(* Logix 5000 project; controller cal1632 1756-L62 rev 16.20; software revision 16.05; part 55 of 57 *)
(* tags used below, declared in another part *)
   FAULT : BOOL;
   p01_recipe_active : recipe;
   p01r02_plc_scan_time_in_sec : REAL;
   p01r09_pb_global_reset : BOOL;
   p29_ao_wdr_turret_selected_speed : REAL;
   p29_di_turret_pos : BOOL;
   p29_di_wdr_index_fwd : BOOL;
   p29_di_wdr_turret : acs800_di_normal;
   p29_di_wt_motor : BOOL;
   p29_do_wdr_turret : acs800_do_normal;
   p29_param_fast_turret_speed : REAL;
   p29_param_slow_turret_speed : REAL;
   p29r15_wdra_active : BOOL;
   p29r16_wdrb_active : BOOL;
   p29r20 : routine;
   p29r20_acc_dec_ramp : SYS_ACC_DEC_RAMP;
   p29r20_accel_rate : REAL;
   p29r20_decel_rate : REAL;
   p29r20_fast_accel : REAL;
   p29r20_fast_decel : REAL;
   p29r20_index_complete : BOOL;
   p29r20_index_move_timer : TIMER;
   p29r20_permissive : BOOL;
   p29r20_request_fwd : BOOL;
   p29r20_request_rev : BOOL;
   p29r20_selected_speed : REAL;
   p29r20_timer_fault : TIMER[10];
   p29r20_timer_warning : TIMER[4];
   p29r20_zero_speed : BOOL;
   p30_di_pin_1 : BOOL;
   p30_di_pin_2 : BOOL;
   p30_di_pin_3 : BOOL;
   p30_di_pin_4 : BOOL;
   p30_di_pin_5 : BOOL;
   p30_di_pin_6 : BOOL;
   p30_di_pin_7 : BOOL;
   p30_di_pin_8 : BOOL;
   p30_di_retraction_down_ls : BOOL;
   p30_di_retraction_up_ls : BOOL;
   p30_di_rotation_fault : BOOL;
   p30_di_ss_close : BOOL;
   p30_di_ss_open : BOOL;
   p30_dint_to_hmi : DINT[16];
   p30r01 : routine;
   p30r02 : routine;
   p30r02_fault_exists : BOOL;
   p30r02_timer_fault : TIMER[4];
   p30r02_timer_warning : TIMER[4];
   p30r02_unack_fault : BOOL;
   p30r02_unack_warning : BOOL;
   p30r02_warning_exists : BOOL;
   p30r03 : routine;
   p30r03_timer_fault : TIMER[4];
   p30r03_timer_warning : TIMER[4];
   p30r04 : routine;
   p30r05 : routine;
   p30r06 : routine;
   p30r07 : routine;
   p30r08 : routine;
   p30r09 : routine;
   p30r10 : routine;
   RETACTION_DELAY_TIMER : TIMER;
   RETRACTION_DELAY_TIMER_2 : TIMER;
(* P29_Winder, continued *)

ROUTINE R20_Winder_Turret_VFD   (* ladder *)
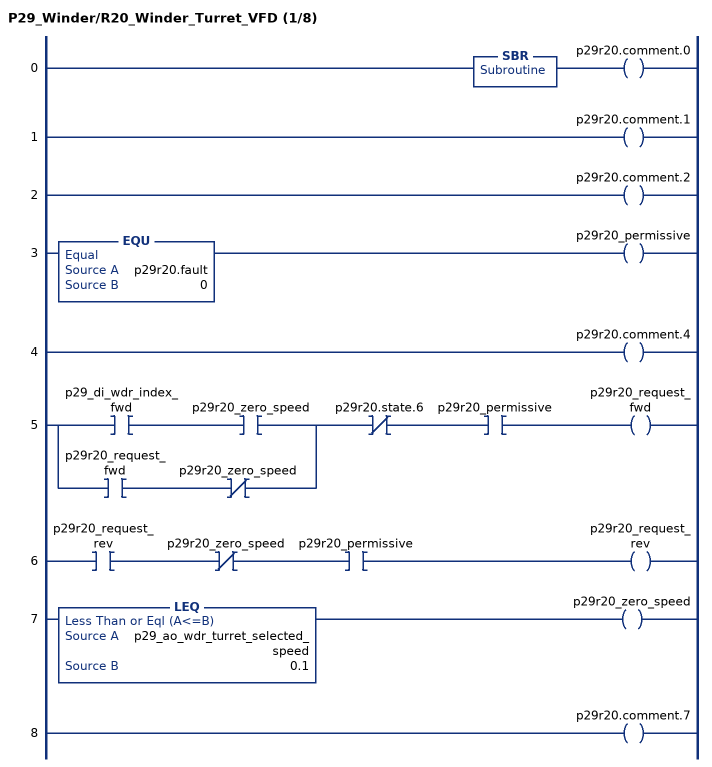
   0: SBR()OTE(p29r20.comment.0);
   1: OTE(p29r20.comment.1);
   2: OTE(p29r20.comment.2);
   3: EQU(p29r20.fault,0)OTE(p29r20_permissive);
   4: OTE(p29r20.comment.4);
   5: [XIC(p29_di_wdr_index_fwd) XIC(p29r20_zero_speed) ,XIC(p29r20_request_fwd) XIO(p29r20_zero_speed) ]XIO(p29r20.state.6)XIC(p29r20_permissive)OTE(p29r20_request_fwd);
   6: XIC(p29r20_request_rev)XIO(p29r20_zero_speed)XIC(p29r20_permissive)OTE(p29r20_request_rev);
   7: LEQ(p29_ao_wdr_turret_selected_speed,0.1)OTE(p29r20_zero_speed);
   8: OTE(p29r20.comment.7);
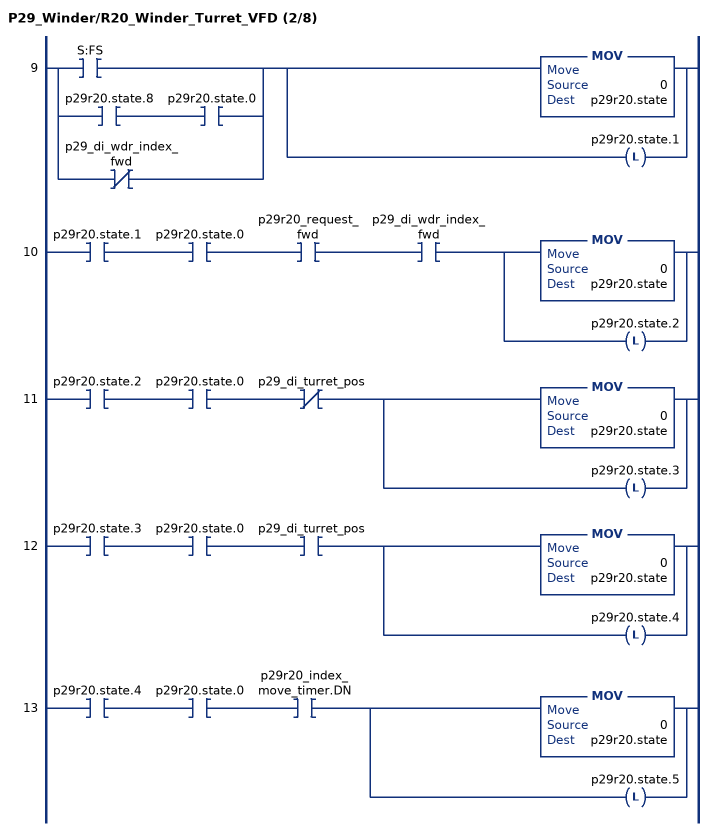
   9: [XIC(S:FS) ,XIC(p29r20.state.8) XIC(p29r20.state.0) ,XIO(p29_di_wdr_index_fwd) ][MOV(0,p29r20.state) ,OTL(p29r20.state.1) ];
   10: XIC(p29r20.state.1)XIC(p29r20.state.0)XIC(p29r20_request_fwd)XIC(p29_di_wdr_index_fwd)[MOV(0,p29r20.state) ,OTL(p29r20.state.2) ];
   11: XIC(p29r20.state.2)XIC(p29r20.state.0)XIO(p29_di_turret_pos)[MOV(0,p29r20.state) ,OTL(p29r20.state.3) ];
   12: XIC(p29r20.state.3)XIC(p29r20.state.0)XIC(p29_di_turret_pos)[MOV(0,p29r20.state) ,OTL(p29r20.state.4) ];
   13: XIC(p29r20.state.4)XIC(p29r20.state.0)XIC(p29r20_index_move_timer.DN)[MOV(0,p29r20.state) ,OTL(p29r20.state.5) ];
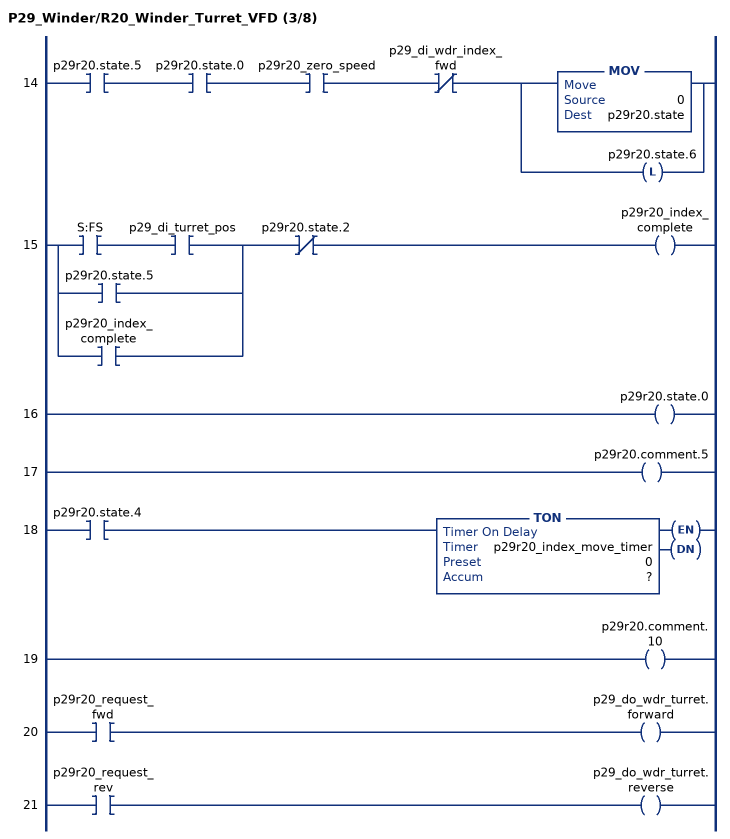
   14: XIC(p29r20.state.5)XIC(p29r20.state.0)XIC(p29r20_zero_speed)XIO(p29_di_wdr_index_fwd)[MOV(0,p29r20.state) ,OTL(p29r20.state.6) ];
   15: [XIC(S:FS) XIC(p29_di_turret_pos) ,XIC(p29r20.state.5) ,XIC(p29r20_index_complete) ]XIO(p29r20.state.2)OTE(p29r20_index_complete);
   16: OTE(p29r20.state.0);
   17: OTE(p29r20.comment.5);
   18: XIC(p29r20.state.4)TON(p29r20_index_move_timer,?,?);
   19: OTE(p29r20.comment.10);
   20: XIC(p29r20_request_fwd)OTE(p29_do_wdr_turret.forward);
   21: XIC(p29r20_request_rev)OTE(p29_do_wdr_turret.reverse);
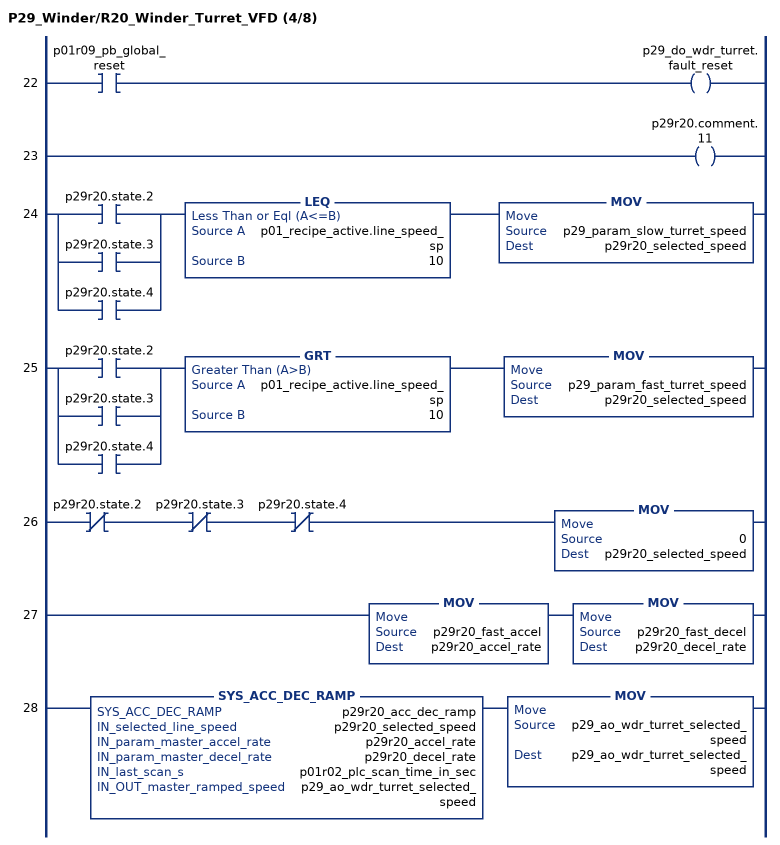
   22: XIC(p01r09_pb_global_reset)OTE(p29_do_wdr_turret.fault_reset);
   23: OTE(p29r20.comment.11);
   24: [XIC(p29r20.state.2) ,XIC(p29r20.state.3) ,XIC(p29r20.state.4) ]LEQ(p01_recipe_active.line_speed_sp,10)MOV(p29_param_slow_turret_speed,p29r20_selected_speed);
   25: [XIC(p29r20.state.2) ,XIC(p29r20.state.3) ,XIC(p29r20.state.4) ]GRT(p01_recipe_active.line_speed_sp,10)MOV(p29_param_fast_turret_speed,p29r20_selected_speed);
   26: XIO(p29r20.state.2)XIO(p29r20.state.3)XIO(p29r20.state.4)MOV(0,p29r20_selected_speed);
   27: MOV(p29r20_fast_accel,p29r20_accel_rate)MOV(p29r20_fast_decel,p29r20_decel_rate);
   28: SYS_ACC_DEC_RAMP(p29r20_acc_dec_ramp,p29r20_selected_speed,p29r20_accel_rate,p29r20_decel_rate,p01r02_plc_scan_time_in_sec,p29_ao_wdr_turret_selected_speed)MOV(p29_ao_wdr_turret_selected_speed,p29_ao_wdr_turret_selected_speed);
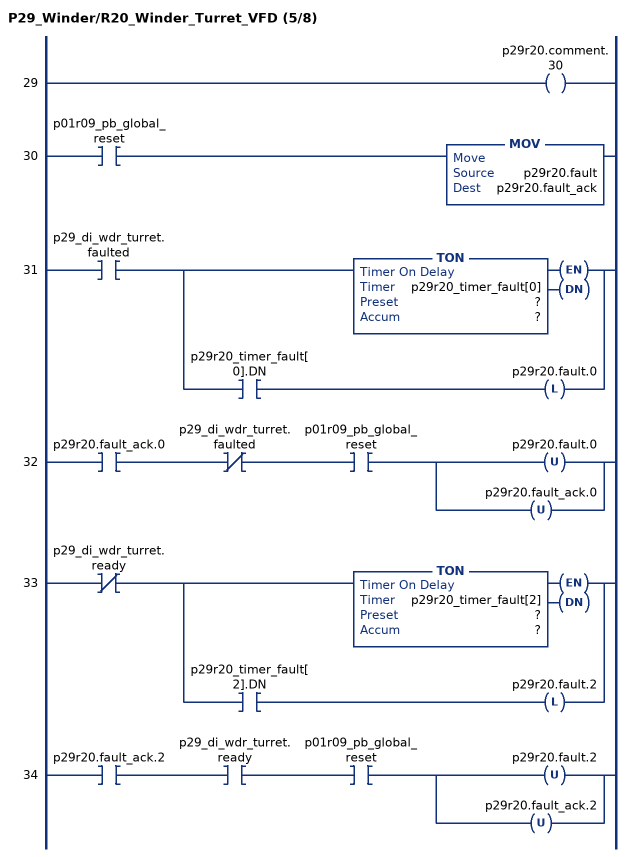
   29: OTE(p29r20.comment.30);
   30: XIC(p01r09_pb_global_reset)MOV(p29r20.fault,p29r20.fault_ack);
   31: XIC(p29_di_wdr_turret.faulted)[TON(p29r20_timer_fault[0],?,?) ,XIC(p29r20_timer_fault[0].DN) OTL(p29r20.fault.0) ];
   32: XIC(p29r20.fault_ack.0)XIO(p29_di_wdr_turret.faulted)XIC(p01r09_pb_global_reset)[OTU(p29r20.fault.0) ,OTU(p29r20.fault_ack.0) ];
   33: XIO(p29_di_wdr_turret.ready)[TON(p29r20_timer_fault[2],?,?) ,XIC(p29r20_timer_fault[2].DN) OTL(p29r20.fault.2) ];
   34: XIC(p29r20.fault_ack.2)XIC(p29_di_wdr_turret.ready)XIC(p01r09_pb_global_reset)[OTU(p29r20.fault.2) ,OTU(p29r20.fault_ack.2) ];
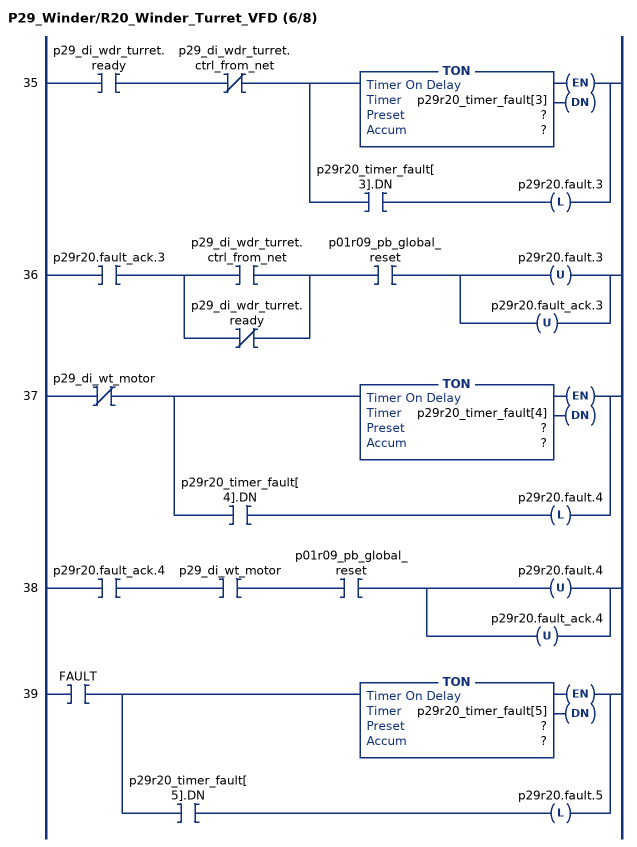
   35: XIC(p29_di_wdr_turret.ready)XIO(p29_di_wdr_turret.ctrl_from_net)[TON(p29r20_timer_fault[3],?,?) ,XIC(p29r20_timer_fault[3].DN) OTL(p29r20.fault.3) ];
   36: XIC(p29r20.fault_ack.3)[XIC(p29_di_wdr_turret.ctrl_from_net) ,XIO(p29_di_wdr_turret.ready) ]XIC(p01r09_pb_global_reset)[OTU(p29r20.fault.3) ,OTU(p29r20.fault_ack.3) ];
   37: XIO(p29_di_wt_motor)[TON(p29r20_timer_fault[4],?,?) ,XIC(p29r20_timer_fault[4].DN) OTL(p29r20.fault.4) ];
   38: XIC(p29r20.fault_ack.4)XIC(p29_di_wt_motor)XIC(p01r09_pb_global_reset)[OTU(p29r20.fault.4) ,OTU(p29r20.fault_ack.4) ];
   39: XIC(FAULT)[TON(p29r20_timer_fault[5],?,?) ,XIC(p29r20_timer_fault[5].DN) OTL(p29r20.fault.5) ];
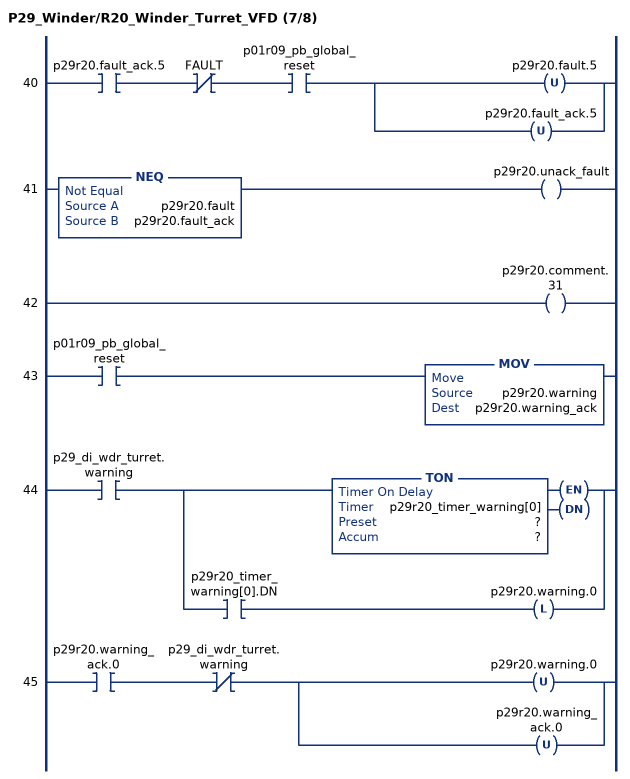
   40: XIC(p29r20.fault_ack.5)XIO(FAULT)XIC(p01r09_pb_global_reset)[OTU(p29r20.fault.5) ,OTU(p29r20.fault_ack.5) ];
   41: NEQ(p29r20.fault,p29r20.fault_ack)OTE(p29r20.unack_fault);
   42: OTE(p29r20.comment.31);
   43: XIC(p01r09_pb_global_reset)MOV(p29r20.warning,p29r20.warning_ack);
   44: XIC(p29_di_wdr_turret.warning)[TON(p29r20_timer_warning[0],?,?) ,XIC(p29r20_timer_warning[0].DN) OTL(p29r20.warning.0) ];
   45: XIC(p29r20.warning_ack.0)XIO(p29_di_wdr_turret.warning)[OTU(p29r20.warning.0) ,OTU(p29r20.warning_ack.0) ];
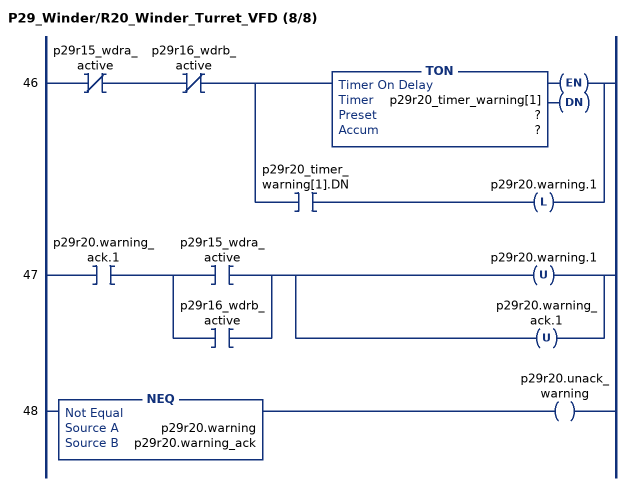
   46: XIO(p29r15_wdra_active)XIO(p29r16_wdrb_active)[TON(p29r20_timer_warning[1],?,?) ,XIC(p29r20_timer_warning[1].DN) OTL(p29r20.warning.1) ];
   47: XIC(p29r20.warning_ack.1)[XIC(p29r15_wdra_active) ,XIC(p29r16_wdrb_active) ][OTU(p29r20.warning.1) ,OTU(p29r20.warning_ack.1) ];
   48: NEQ(p29r20.warning,p29r20.warning_ack)OTE(p29r20.unack_warning);
END_ROUTINE
END_PROGRAM

PROGRAM P30_Retraction_System   (* main routine R01_Main *)

ROUTINE R01_Main   (* ladder *)
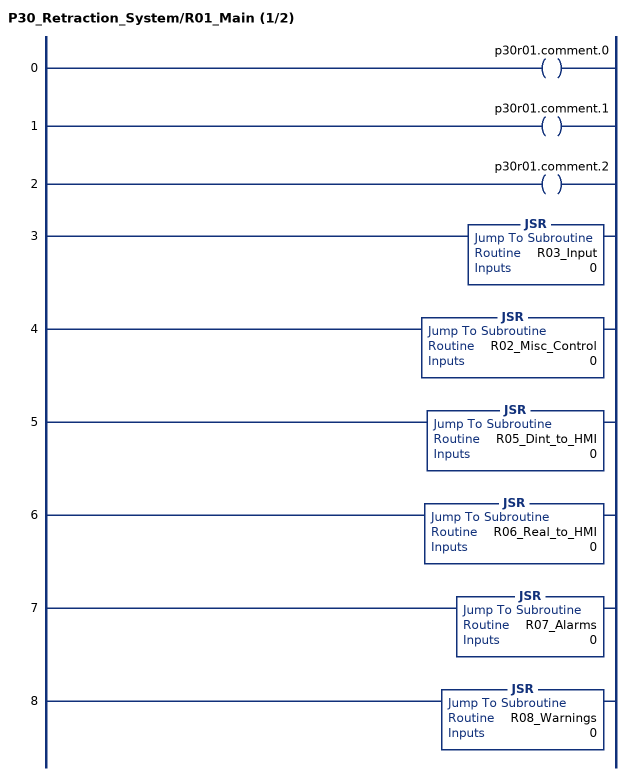
   0: OTE(p30r01.comment.0);
   1: OTE(p30r01.comment.1);
   2: OTE(p30r01.comment.2);
   3: JSR(R03_Input,0);
   4: JSR(R02_Misc_Control,0);
   5: JSR(R05_Dint_to_HMI,0);
   6: JSR(R06_Real_to_HMI,0);
   7: JSR(R07_Alarms,0);
   8: JSR(R08_Warnings,0);
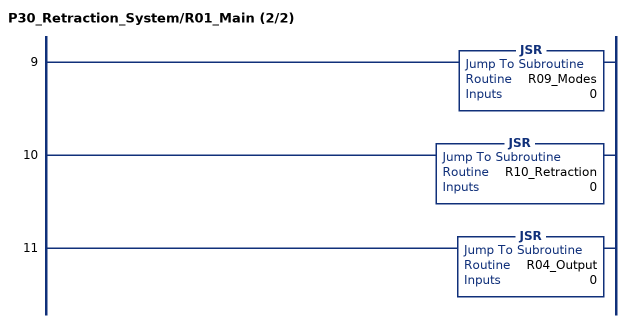
   9: JSR(R09_Modes,0);
   10: JSR(R10_Retraction,0);
   11: JSR(R04_Output,0);
END_ROUTINE

ROUTINE R02_Misc_Control   (* ladder *)
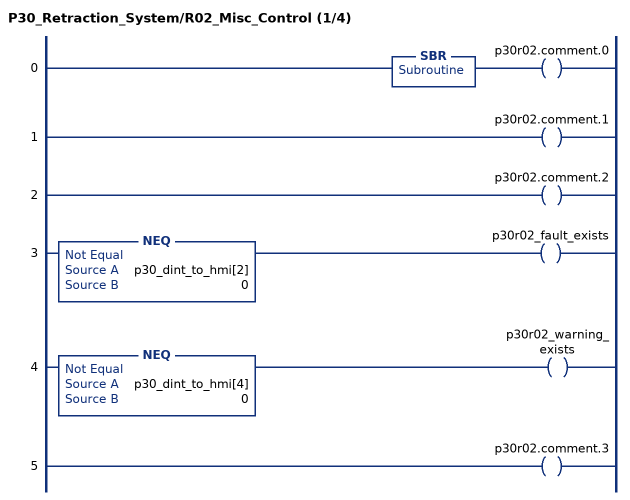
   0: SBR()OTE(p30r02.comment.0);
   1: OTE(p30r02.comment.1);
   2: OTE(p30r02.comment.2);
   3: NEQ(p30_dint_to_hmi[2],0)OTE(p30r02_fault_exists);
   4: NEQ(p30_dint_to_hmi[4],0)OTE(p30r02_warning_exists);
   5: OTE(p30r02.comment.3);
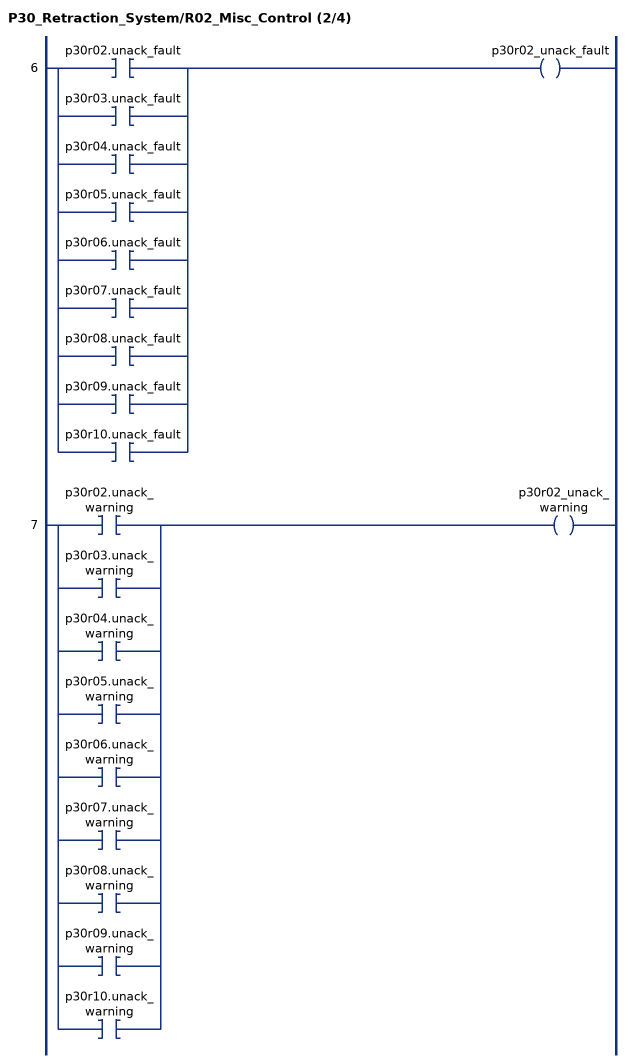
   6: [XIC(p30r02.unack_fault) ,XIC(p30r03.unack_fault) ,XIC(p30r04.unack_fault) ,XIC(p30r05.unack_fault) ,XIC(p30r06.unack_fault) ,XIC(p30r07.unack_fault) ,XIC(p30r08.unack_fault) ,XIC(p30r09.unack_fault) ,XIC(p30r10.unack_fault) ]OTE(p30r02_unack_fault);
   7: [XIC(p30r02.unack_warning) ,XIC(p30r03.unack_warning) ,XIC(p30r04.unack_warning) ,XIC(p30r05.unack_warning) ,XIC(p30r06.unack_warning) ,XIC(p30r07.unack_warning) ,XIC(p30r08.unack_warning) ,XIC(p30r09.unack_warning) ,XIC(p30r10.unack_warning) ]OTE(p30r02_unack_warning);
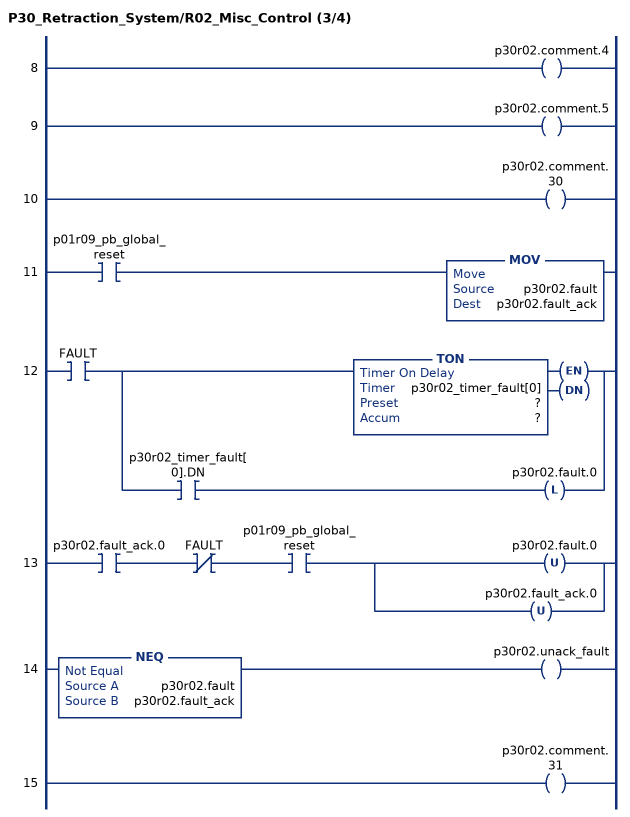
   8: OTE(p30r02.comment.4);
   9: OTE(p30r02.comment.5);
   10: OTE(p30r02.comment.30);
   11: XIC(p01r09_pb_global_reset)MOV(p30r02.fault,p30r02.fault_ack);
   12: XIC(FAULT)[TON(p30r02_timer_fault[0],?,?) ,XIC(p30r02_timer_fault[0].DN) OTL(p30r02.fault.0) ];
   13: XIC(p30r02.fault_ack.0)XIO(FAULT)XIC(p01r09_pb_global_reset)[OTU(p30r02.fault.0) ,OTU(p30r02.fault_ack.0) ];
   14: NEQ(p30r02.fault,p30r02.fault_ack)OTE(p30r02.unack_fault);
   15: OTE(p30r02.comment.31);
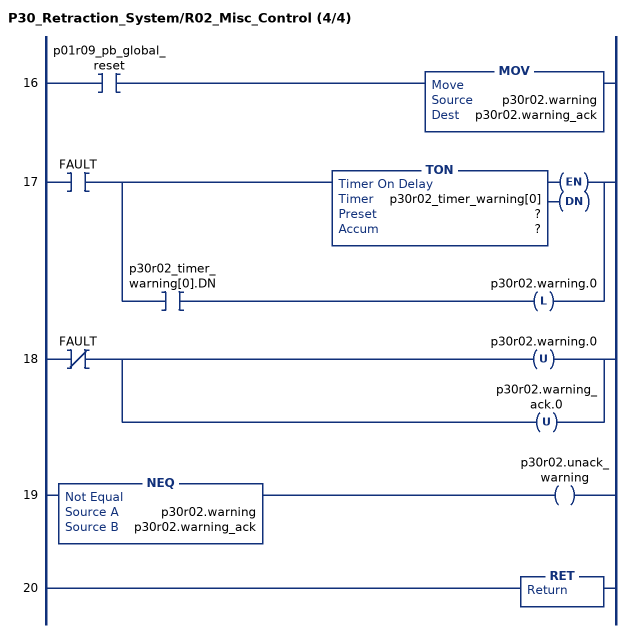
   16: XIC(p01r09_pb_global_reset)MOV(p30r02.warning,p30r02.warning_ack);
   17: XIC(FAULT)[TON(p30r02_timer_warning[0],?,?) ,XIC(p30r02_timer_warning[0].DN) OTL(p30r02.warning.0) ];
   18: XIO(FAULT)[OTU(p30r02.warning.0) ,OTU(p30r02.warning_ack.0) ];
   19: NEQ(p30r02.warning,p30r02.warning_ack)OTE(p30r02.unack_warning);
   20: RET();
END_ROUTINE

ROUTINE R03_Input   (* ladder *)
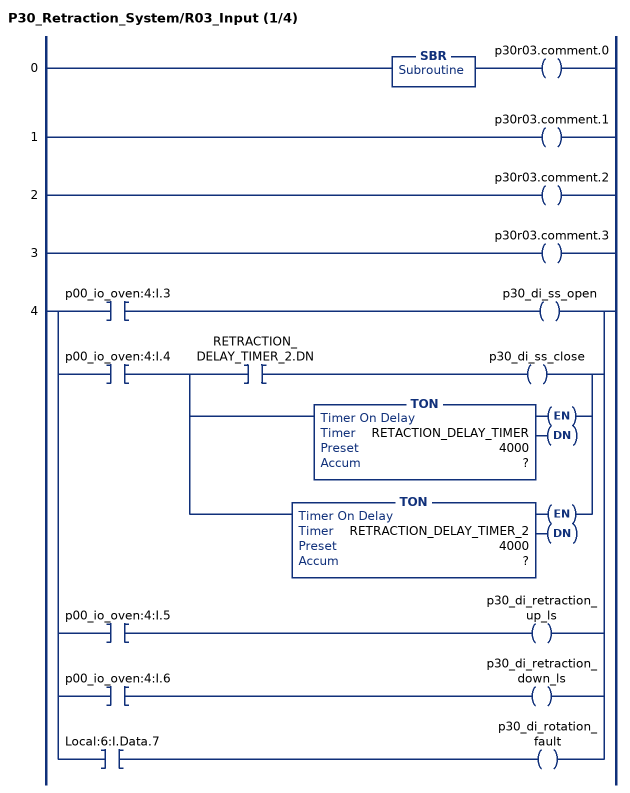
   0: SBR()OTE(p30r03.comment.0);
   1: OTE(p30r03.comment.1);
   2: OTE(p30r03.comment.2);
   3: OTE(p30r03.comment.3);
   4: [XIC(p00_io_oven:4:I.3) OTE(p30_di_ss_open) ,XIC(p00_io_oven:4:I.4) [XIC(RETRACTION_DELAY_TIMER_2.DN) OTE(p30_di_ss_close) ,TON(RETACTION_DELAY_TIMER,?,?) ,TON(RETRACTION_DELAY_TIMER_2,?,?) ] ,XIC(p00_io_oven:4:I.5) OTE(p30_di_retraction_up_ls) ,XIC(p00_io_oven:4:I.6) OTE(p30_di_retraction_down_ls) ,XIC(Local:6:I.Data.7) OTE(p30_di_rotation_fault) ];
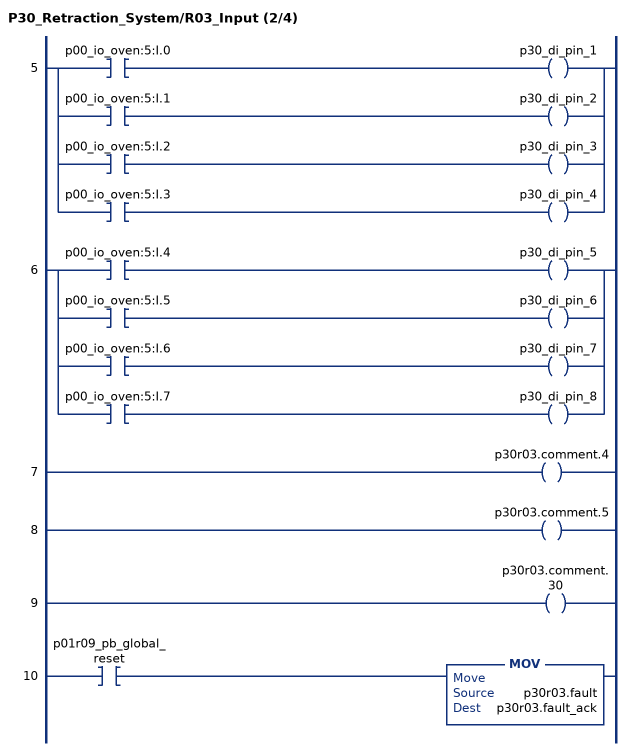
   5: [XIC(p00_io_oven:5:I.0) OTE(p30_di_pin_1) ,XIC(p00_io_oven:5:I.1) OTE(p30_di_pin_2) ,XIC(p00_io_oven:5:I.2) OTE(p30_di_pin_3) ,XIC(p00_io_oven:5:I.3) OTE(p30_di_pin_4) ];
   6: [XIC(p00_io_oven:5:I.4) OTE(p30_di_pin_5) ,XIC(p00_io_oven:5:I.5) OTE(p30_di_pin_6) ,XIC(p00_io_oven:5:I.6) OTE(p30_di_pin_7) ,XIC(p00_io_oven:5:I.7) OTE(p30_di_pin_8) ];
   7: OTE(p30r03.comment.4);
   8: OTE(p30r03.comment.5);
   9: OTE(p30r03.comment.30);
   10: XIC(p01r09_pb_global_reset)MOV(p30r03.fault,p30r03.fault_ack);
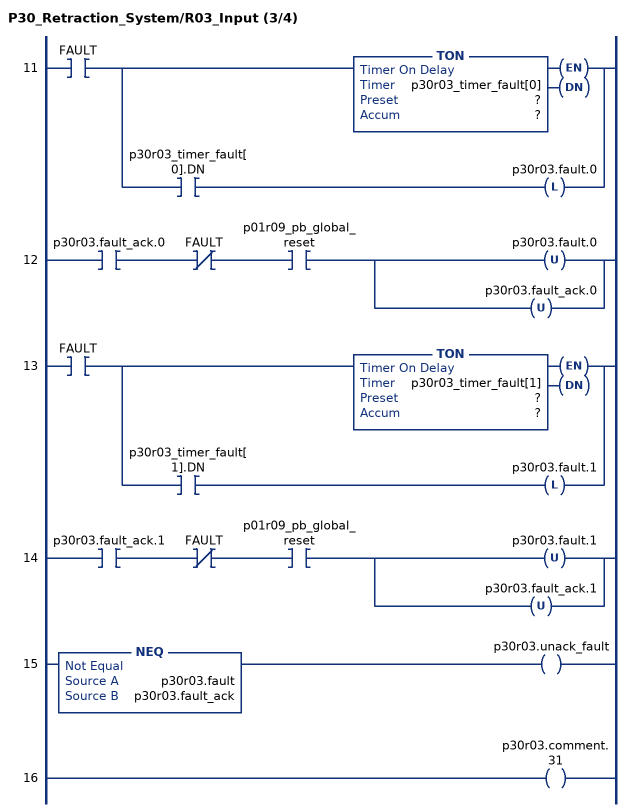
   11: XIC(FAULT)[TON(p30r03_timer_fault[0],?,?) ,XIC(p30r03_timer_fault[0].DN) OTL(p30r03.fault.0) ];
   12: XIC(p30r03.fault_ack.0)XIO(FAULT)XIC(p01r09_pb_global_reset)[OTU(p30r03.fault.0) ,OTU(p30r03.fault_ack.0) ];
   13: XIC(FAULT)[TON(p30r03_timer_fault[1],?,?) ,XIC(p30r03_timer_fault[1].DN) OTL(p30r03.fault.1) ];
   14: XIC(p30r03.fault_ack.1)XIO(FAULT)XIC(p01r09_pb_global_reset)[OTU(p30r03.fault.1) ,OTU(p30r03.fault_ack.1) ];
   15: NEQ(p30r03.fault,p30r03.fault_ack)OTE(p30r03.unack_fault);
   16: OTE(p30r03.comment.31);
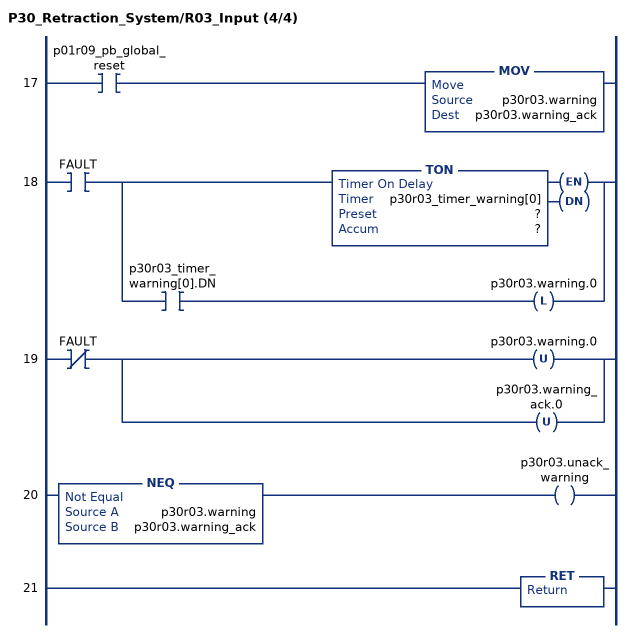
   17: XIC(p01r09_pb_global_reset)MOV(p30r03.warning,p30r03.warning_ack);
   18: XIC(FAULT)[TON(p30r03_timer_warning[0],?,?) ,XIC(p30r03_timer_warning[0].DN) OTL(p30r03.warning.0) ];
   19: XIO(FAULT)[OTU(p30r03.warning.0) ,OTU(p30r03.warning_ack.0) ];
   20: NEQ(p30r03.warning,p30r03.warning_ack)OTE(p30r03.unack_warning);
   21: RET();
END_ROUTINE
